(* Logix 5000 project; controller KTC_ball vendor 1 type 14 code 92 rev 30.11; software revision 30.00 *)

TASK MainTask (continuous, watchdog 500 ms) : MainProgram

MODULES
   Local : vendor 1 type 14 code 92 (ICP 0, rev 30.11)
END_MODULES

PROGRAM MainProgram   (* main routine MainRoutine *)

ROUTINE MainRoutine   (* ladder *)
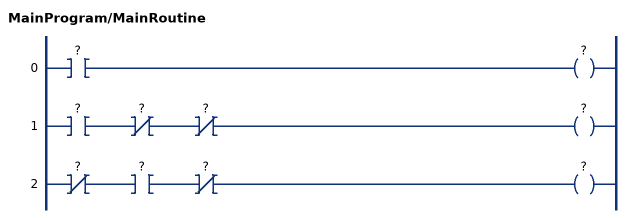
   0: XIC(?)OTE(?);
   1: XIC(?)XIO(?)XIO(?)OTE(?);
   2: XIO(?)XIC(?)XIO(?)OTE(?);
END_ROUTINE
END_PROGRAM
